FUNCTION_BLOCK NF_Logic
VAR
	_piston : TcoPneumatics.Cylinder(NF_MAIN.Context);
END_VAR


_piston.Service();

_piston();

END_FUNCTION_BLOCK

(* stored: Version 1.1.0.1, ProductVersion 3.1.4024.6
   POU NF_Logic: Id {a15ad3d6-c3ee-43f1-a95a-15ff90bf4019}, SpecialFunc None *)
